FUNCTION_BLOCK BinArg IMPLEMENTS I_MutBinArg
VAR
	_val			: LWORD;
END_VAR

PROPERTY Val : LWORD
GET
Val := _val;
END_GET
SET
_val := Val;
END_SET
END_PROPERTY

END_FUNCTION_BLOCK

(* stored: Version 1.1.0.1
   POU BinArg: Id {cb0fcc97-6bd1-4da2-ad95-d55933bfe94a}, SpecialFunc None
   Property Val: Id {561e9447-a720-49d7-897e-fa3dc653c48d}
   Get Get: Id {e19392a7-d96c-4409-af36-6659fa831215}
   Set Set: Id {92426485-401c-4221-a784-58afae172b3e} *)
